FUNCTION_BLOCK TwoCars
  (* Standard: 61499-2 *)
  (* Version 0.1, 2015-00-08, SYY, SYY-PC *)
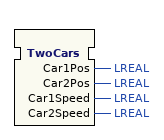
  VAR_OUTPUT
    Car1Pos : LREAL;
    Car2Pos : LREAL;
    Car1Speed : LREAL;
    Car2Speed : LREAL;
  END_VAR
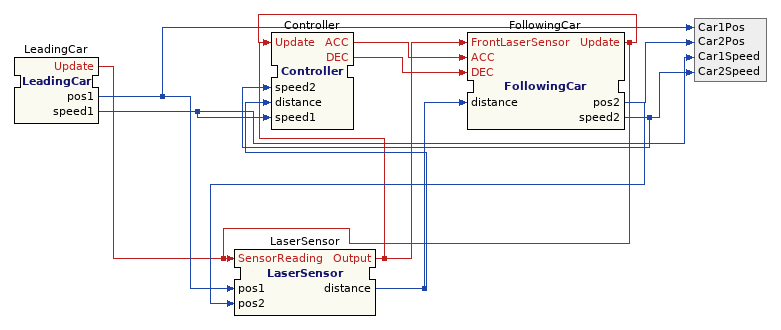
  FBS
    LeadingCar : LeadingCar;
    FollowingCar : FollowingCar;
    LaserSensor : LaserSensor;
    Controller : Controller;
  END_FBS
  EVENT_CONNECTIONS
    LeadingCar.Update TO LaserSensor.SensorReading;
    FollowingCar.Update TO LaserSensor.SensorReading;
    FollowingCar.Update TO Controller.Update;
    LaserSensor.Output TO FollowingCar.FrontLaserSensor;
    LaserSensor.Output TO Controller.Update;
    Controller.ACC TO FollowingCar.ACC;
    Controller.DEC TO FollowingCar.DEC;
  END_CONNECTIONS
  DATA_CONNECTIONS
    LeadingCar.pos1 TO Car1Pos;
    FollowingCar.pos2 TO Car2Pos;
    LeadingCar.speed1 TO Car1Speed;
    FollowingCar.speed2 TO Car2Speed;
    LeadingCar.pos1 TO LaserSensor.pos1;
    LeadingCar.speed1 TO Controller.speed1;
    FollowingCar.pos2 TO LaserSensor.pos2;
    FollowingCar.speed2 TO Controller.speed2;
    LaserSensor.distance TO FollowingCar.distance;
    LaserSensor.distance TO Controller.distance;
  END_CONNECTIONS
END_FUNCTION_BLOCK
